(* Schneider Machine Expert - Basic project diagrama_ladder, file version 2.8.0.0 *)
(* ProjectInformations: Name=SEQUENCIA DE ATUADORES: A+B+A-B- *)
(* UserInformations: LastName=GAGLIANO, FirstName=LEONARDO *)

HARDWARE
  Cpu 0: TM221CE40T
  EthernetConfiguration: NetworkName=M221, IpAllocationMode=FixedAddress, IpAddress=0.0.0.0, SubnetMask=0.0.0.0
  SerialLineConfiguration: Baud=Baud19200, Parity=ParityEven, DataBits=DataBits8, StopBits=StopBits1, PhysicalMedium=PhysicalMediumRs485, TransmissionMode=TransmissionModeModbusRtu, SlaveId=1, Addressing=SlaveAddressing
  MastTask: UsePeriodScanMode=false, PeriodScan=100
  FastTask: Period=255
  CpuBehavior: StartingMode=StartAsPreviousState, AutoSaveRamOnEeprom=true, WatchdogPeriod=250

SYMBOLS  (address, symbol, comment, settings)
  %M0         "A+"
  %M1         "B+"
  %M2         "A-"
  %M3         "B-"
  %M4         "COND_RESET"
  %I0.0     I0  "B0"
  %I0.1     I1  "S1"
  %I0.2     I2  "S2"
  %I0.3     I3  "S3"
  %I0.4     I4  "S4"
  %Q0.0     Q0
  %Q0.1     Q1

POU Novo POU
  (* SectionNumber=1 *)

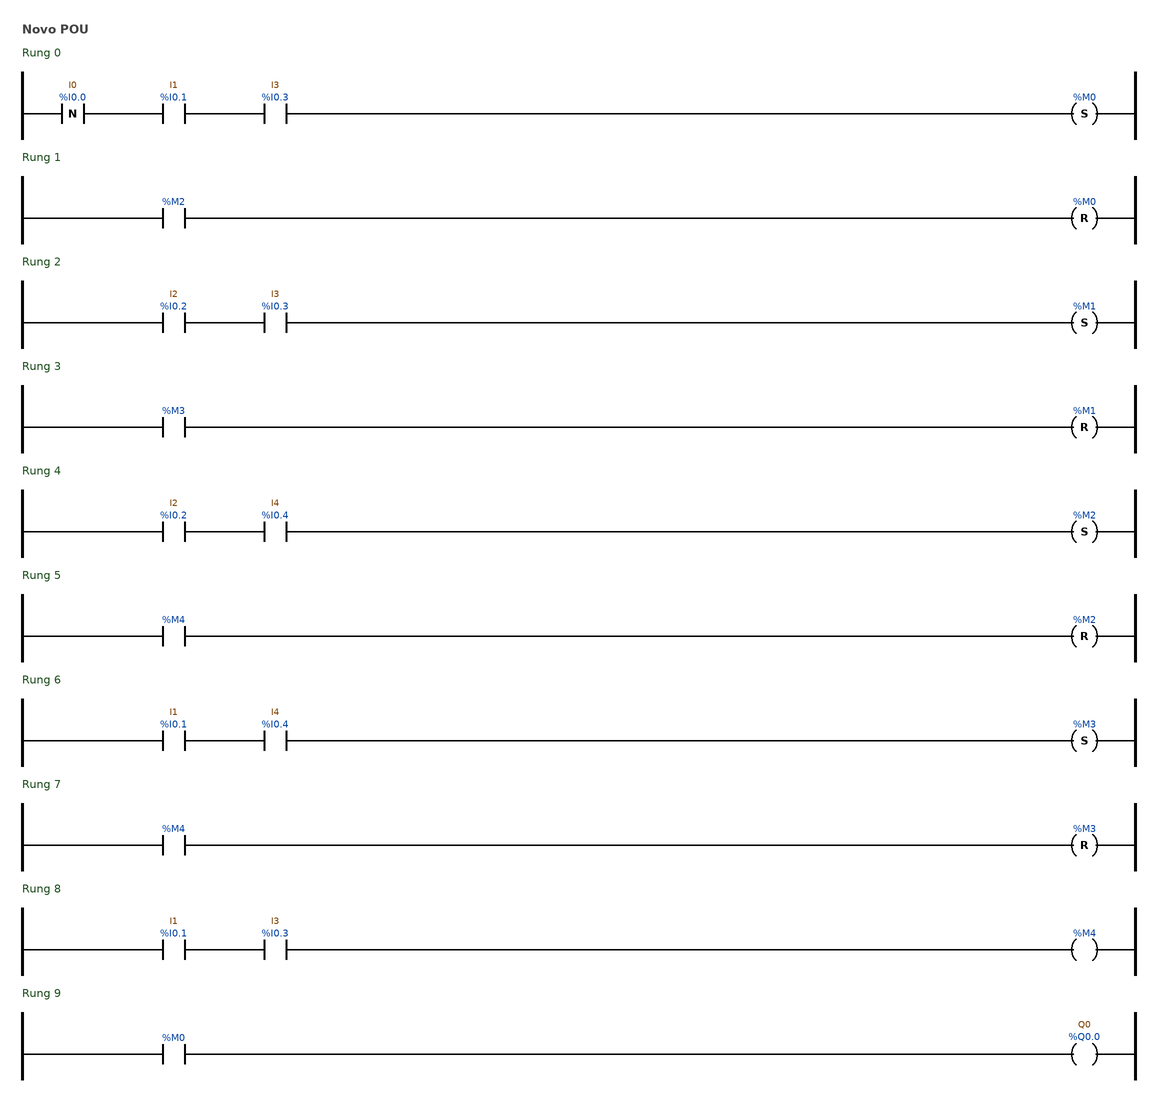

// Rung 0
  LDF %I0.0               (* I0 *)
  AND %I0.1               (* I1 *)
  AND %I0.3               (* I3 *)
  S %M0
  // as ST:
  //   IF FALLING(I0) AND I1 AND I3 THEN %M0 := TRUE; END_IF;

// Rung 1
  LD %M2
  R %M0
  // as ST:
  //   IF %M2 THEN %M0 := FALSE; END_IF;

// Rung 2
  LD %I0.2                (* I2 *)
  AND %I0.3               (* I3 *)
  S %M1
  // as ST:
  //   IF I2 AND I3 THEN %M1 := TRUE; END_IF;

// Rung 3
  LD %M3
  R %M1
  // as ST:
  //   IF %M3 THEN %M1 := FALSE; END_IF;

// Rung 4
  LD %I0.2                (* I2 *)
  AND %I0.4               (* I4 *)
  S %M2
  // as ST:
  //   IF I2 AND I4 THEN %M2 := TRUE; END_IF;

// Rung 5
  LD %M4
  R %M2
  // as ST:
  //   IF %M4 THEN %M2 := FALSE; END_IF;

// Rung 6
  LD %I0.1                (* I1 *)
  AND %I0.4               (* I4 *)
  S %M3
  // as ST:
  //   IF I1 AND I4 THEN %M3 := TRUE; END_IF;

// Rung 7
  LD %M4
  R %M3
  // as ST:
  //   IF %M4 THEN %M3 := FALSE; END_IF;

// Rung 8
  LD %I0.1                (* I1 *)
  AND %I0.3               (* I3 *)
  ST %M4
  // as ST:
  //   %M4 := I1 AND I3;

// Rung 9
  LD %M0
  ST %Q0.0                (* Q0 *)
  // as ST:
  //   Q0 := %M0;

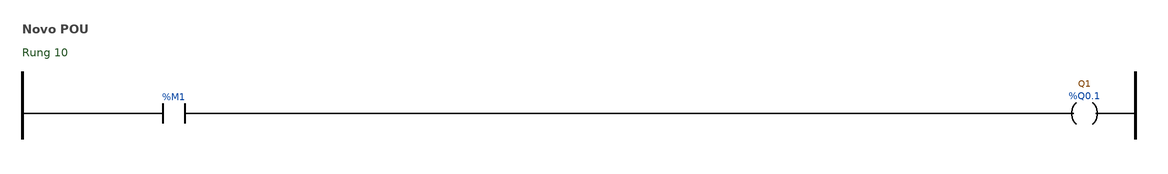

// Rung 10
  LD %M1
  ST %Q0.1                (* Q1 *)
  // as ST:
  //   Q1 := %M1;
